KUKA KRL data list: Weld_PartA.dat

&ACCESS RV
&REL 1
DEFDAT Weld_PartA PUBLIC
  DECL E6POS HOME={A1 0.0, A2 -90.0, A3 90.0, A4 0.0, A5 0.0, A6 0.0}
  DECL E6POS P1={X 400.0, Y 100.0, Z 250.0, A 0.0, B 90.0, C 0.0, S 2, T 10}
  DECL E6POS P2={X 400.0, Y 300.0, Z 250.0, A 0.0, B 90.0, C 0.0, S 2, T 10}
  DECL E6POS P3={X 400.0, Y 500.0, Z 250.0, A 0.0, B 90.0, C 0.0, S 2, T 10}
ENDDAT
